(* CODESYS project Elevator.project

Project tree, tasks and I/O mapping:
  Device : Elmo Platinum Maestro, Elmo Motion Control, version 1.0.0.2
    application Application
      libraries: Standard, * (System); VisuDialogs, * (System)
      task MainTask (cyclic, interval t#20ms, priority 1) calls PLC_PRG
      task VISU_TASK (cyclic, interval 100 ms, priority 31) calls VisuElems.Visu_Prg
      program PLC_PRG [ST]
      visualisation Visualization
      visualisation Elevator
      01_Enumerator/
        data type eFloor
      02_Structure/
        data type stElevator
        data type stFloor
      03_Module/
        function block FB_Elevator [ST]: M_SpecialFloorSelect, pSpecialFloor, M_DoorStatus, M_ElevatorType, M_FindFloor, M_ElevatorMove, M_ElevatorSelect, M_ElevatorButtonDisable, M_FloorMove
        function block FB_FreightElevator [ST]: pSpecialFloor
        function block FB_Floor [ST]
        function F_RandElevator [ST]
      04_Component/
      visualisation Floor
      global variables GVL_Random
    Elmo_Master_Device : Elmo Master Device, Elmo, version 1.0.0.2
  libraries: VisuSymbols, 3.5.10.0 (System)
  text list GlobalTextList
*)

// Device/Application/02_Structure/stElevator
TYPE stElevator :
STRUCT
	sElMove: STRING;
	xFloor1: BOOL;
	
	xFloor2: BOOL;
	
	xFloor3: BOOL;
	
	xFloor4: BOOL;
	
	xFloor5: BOOL;
	
	xSpecialFloor: BOOL;
	xSpecialLight: BOOL;
	sSpecialFloorText: STRING;
	xInvisibleLamp: BOOL;
	
	xOpen: BOOL;
	xClose: BOOL;
	sDoorStatus: STRING;
	//trig_Door: r_trig;
	//trig_CloseDoor: r_trig;
	sElevatorType: STRING;
	iElevatorMove: INT;
	
	sElevatorFloor: STRING;
END_STRUCT
END_TYPE

// Device/Application/02_Structure/stFloor
TYPE stFloor :
STRUCT
	sFloor: STRING;
	iPeople: INT;
	iPeopleCurrent: INT;
	xCall: BOOL;
END_STRUCT
END_TYPE

// Device/Application/01_Enumerator/eFloor
{attribute 'qualified_only'}
{attribute 'strict'}
TYPE eFloor :
(
	F1 := 0,
	F2 := -475,
	F3 := -935,
	F4 := -1375,
	F5 := -1800
);
END_TYPE

// Device/Application/GVL_Random
{attribute 'qualified_only'}
VAR_GLOBAL
	g_seed : INT := 107;
END_VAR

// Device/Application/PLC_PRG
PROGRAM PLC_PRG
VAR
	stFloorData: ARRAY[1..uiFloors] OF stFloor;
	fbFloor: ARRAY[1..uiFloors] OF FB_Floor;
	iFloor: INT;
	stFreightFloor: stFloor;
	iRandFloor: int;
	
	stElevatorData: ARRAY[1..uiElevators] OF stElevator;
	fbElevator: ARRAY[1..uiElevators] OF FB_Elevator;
	iElevator: INT;
	stFreightElevator: stElevator;
	fbFreightElevator: FB_FreightElevator;
	
	xRandElevator: BOOL;
END_VAR

VAR CONSTANT
	uiFloors: UINT:= 5;
	uiElevators: UINT:= 3;
END_VAR

FOR iFloor:=1 TO uiFloors BY 1 DO
	stFloorData[iFloor].sFloor := concat(str1:='F',str2:=INT_TO_STRING(iFloor));
	stFloorData[iFloor].iPeopleCurrent := stFloorData[iFloor].iPeople;
	
	//IF stFloorData[iFloor].xCall = TRUE THEN
		//iRandFloor := F_RandElevator();
		//stElevatorData[iRandFloor]
		//IF NOT xRandElevator THEN
			//iRandFloor := F_RandElevator();
			//xRandElevator := TRUE;
		//END_IF
		iRandFloor := fbElevator[iFloor].M_ElevatorSelect(is_Floor := stFloorData[iFloor].sFloor,ist_Elevator:=stElevatorData);
		//stElevatorData[iRandFloor].sElMove := fbElevator[iRandFloor].os_ElMove;
		fbElevator[iRandFloor].M_ElevatorMove(is_Floor := stFloorData[iFloor].sFloor,iElMove := stElevatorData[iRandFloor].iElevatorMove,xElevatorMove := stFloorData[iFloor].xCall);
		//stFloorData[iFloor].xCall := FALSE;
	//END_IF
END_FOR

stFreightFloor.sFloor := 'B1';
stFreightFloor.iPeopleCurrent := stFreightFloor.iPeople;
//iRandFloor := F_RandElevator();


FOR iElevator:= 1 TO uiElevators BY 1 DO
	
    stElevatorData[iElevator].sElMove := fbElevator[iElevator].os_ElMove;
	stElevatorData[iElevator].sSpecialFloorText := fbElevator[iElevator].pSpecialFloor;
	fbElevator[iElevator].ix_FloorButton := stElevatorData[iElevator].xSpecialFloor;
	stElevatorData[iElevator].xSpecialLight := fbElevator[iElevator].M_SpecialFloorSelect();
	
	fbElevator[iElevator].M_DoorStatus(ix_Open:=stElevatorData[iElevator].xOpen,ix_Close:= stElevatorData[iElevator].xClose);
	stElevatorData[iElevator].sDoorStatus := fbElevator[iElevator].os_DoorStatus;
	stElevatorData[iElevator].xOpen := fbElevator[iElevator].ox_Door;
	stElevatorData[iElevator].xClose := NOT fbElevator[iElevator].ox_Door;
	fbElevator[iElevator].M_ElevatorType(is_SpecialFloorText:= stElevatorData[iElevator].sSpecialFloorText);
	stElevatorData[iElevator].sElevatorType := fbElevator[iElevator].os_ElevatorType;
	//IF(stElevatorData[iElevator].iElevatorMove <> -1800) THEN
	  //stElevatorData[iElevator].iElevatorMove := stElevatorData[iElevator].iElevatorMove-1;
    //END_IF
	//IF(stElevatorData[iElevator].xFloor1 = TRUE) THEN
		//IF stElevatorData[iElevator].iElevatorMove < -475 THEN
	      //stElevatorData[iElevator].iElevatorMove := stElevatorData[iElevator].iElevatorMove+1;
        //END_IF

        //IF stElevatorData[iElevator].iElevatorMove > -475 THEN
	      //stElevatorData[iElevator].iElevatorMove := stElevatorData[iElevator].iElevatorMove-1;
        //END_IF
	//END_IF
	fbElevator[iElevator].M_ElevatorButtonDisable(xF1:= stElevatorData[iElevator].xFloor1, xF2:= stElevatorData[iElevator].xFloor2, xF3:= stElevatorData[iElevator].xFloor3, xF4:= stElevatorData[iElevator].xFloor4, xF5:= stElevatorData[iElevator].xFloor5);
	fbElevator[iElevator].M_FloorMove(xFloorButton := stElevatorData[iElevator].xFloor1,is_Floor:= 'F1',iElMove := stElevatorData[iElevator].iElevatorMove);
	fbElevator[iElevator].M_FloorMove(xFloorButton := stElevatorData[iElevator].xFloor2,is_Floor:= 'F2',iElMove := stElevatorData[iElevator].iElevatorMove);
	fbElevator[iElevator].M_FloorMove(xFloorButton := stElevatorData[iElevator].xFloor3,is_Floor:= 'F3',iElMove := stElevatorData[iElevator].iElevatorMove);
	fbElevator[iElevator].M_FloorMove(xFloorButton := stElevatorData[iElevator].xFloor4,is_Floor:= 'F4',iElMove := stElevatorData[iElevator].iElevatorMove);
	fbElevator[iElevator].M_FloorMove(xFloorButton := stElevatorData[iElevator].xFloor5,is_Floor:= 'F5',iElMove := stElevatorData[iElevator].iElevatorMove);
	stElevatorData[iElevator].sElevatorFloor := fbElevator[iElevator].M_FindFloor(iElMove:= stElevatorData[iElevator].iElevatorMove);
	
END_FOR

stFreightElevator.sSpecialFloorText := fbFreightElevator.pSpecialFloor;
stFreightElevator.xInvisibleLamp := TRUE;
fbFreightElevator.M_DoorStatus(ix_Open:=stFreightElevator.xOpen,ix_Close:= stFreightElevator.xClose);
stFreightElevator.sDoorStatus := fbFreightElevator.os_DoorStatus;
stFreightElevator.xOpen := fbFreightElevator.ox_Door;
stFreightElevator.xClose := NOT fbFreightElevator.ox_Door;
fbFreightElevator.M_ElevatorType(is_SpecialFloorText:= stFreightElevator.sSpecialFloorText);
stFreightElevator.sElevatorType := fbFreightElevator.os_ElevatorType;
//IF(stFreightElevator.iElevatorMove <> -1400) THEN
	//stFreightElevator.iElevatorMove := stFreightElevator.iElevatorMove-1;
//END_IF

END_PROGRAM

// Device/Application/03_Module/F_RandElevator
FUNCTION F_RandElevator : INT
VAR_INPUT
END_VAR
VAR
END_VAR

GVL_Random.g_seed := GVL_Random.g_seed * 41 + 17;

IF GVL_Random.g_seed < 0 THEN
    GVL_Random.g_seed := -GVL_Random.g_seed;
END_IF;

F_RandElevator := (GVL_Random.g_seed MOD 3) + 1;

END_FUNCTION

// Device/Application/03_Module/FB_Floor
FUNCTION_BLOCK FB_Floor
VAR_INPUT
END_VAR
VAR_OUTPUT
END_VAR
VAR
END_VAR

END_FUNCTION_BLOCK

// Device/Application/03_Module/FB_Elevator
FUNCTION_BLOCK FB_Elevator
VAR_INPUT
	ix_FloorButton: BOOL;
	ix_Open: BOOL;
	ix_Close: BOOL;
	is_SpecialFloorText: STRING;
	iElMove: INT;
	is_Floor: STRING;
END_VAR
VAR_OUTPUT
	ox_FloorLight: BOOL;
	ox_Door: BOOL;
	os_DoorStatus: STRING;
	os_ElevatorType: STRING;
	os_ElMove: STRING;
END_VAR
VAR
	sSpecialFloorText: STRING;
	trig_Door: r_trig;
	trig_CloseDoor: r_trig;
	iChangeString: INT;
	iFloorValue: eFloor;
	xElevatorMove: BOOL;
	a:INT;
	b:INT;
	c:INT;
	
	d1:INT;
	d2:INT;
	d3:INT;
	mindiff: INT;
	req: INT;
	xFloorButton: BOOL;
	xF1: BOOL;
	xF2: BOOL;
	xF3: BOOL;
	xF4: BOOL;
	xF5: BOOL;
END_VAR

METHOD M_SpecialFloorSelect : BOOL
VAR_INPUT
END_VAR
IF ix_FloorButton=TRUE THEN
	M_SpecialFloorSelect := TRUE;
ELSE
	M_SpecialFloorSelect := FALSE;
END_IF
END_METHOD

PROPERTY pSpecialFloor : STRING
GET
pSpecialFloor := 'EMG';
END_GET
END_PROPERTY

METHOD M_DoorStatus : BOOL
VAR_INPUT
	ix_Open: BOOL;
	ix_Close: BOOL;
END_VAR
trig_Door(clk:=ix_Open);
trig_CloseDoor(clk:=ix_Close);

IF trig_CloseDoor.Q THEN
	ox_Door := FALSE;
ELSIF trig_Door.Q THEN
	ox_Door:= TRUE;
END_IF

IF ox_Door THEN
	os_DoorStatus := 'OPEN';
ELSE
	os_DoorStatus := 'CLOSED';
END_IF
END_METHOD

METHOD M_ElevatorType : STRING
VAR_INPUT
	is_SpecialFloorText: STRING;
END_VAR
IF is_SpecialFloorText = 'EMG' THEN
	os_ElevatorType := 'Max 3 People';
ELSIF is_SpecialFloorText = 'B1' THEN
	os_ElevatorType := 'Max 5 People';
END_IF
END_METHOD

METHOD M_FindFloor : STRING
VAR_INPUT
	iElMove: INT;
END_VAR
IF iElMove <= 0 AND iElMove >= -150 THEN
	M_FindFloor := 'F1';

ELSIF iElMove <= -475 AND iElMove >= -650 THEN
	M_FindFloor := 'F2';

ELSIF iElMove <= -935 AND iElMove >= -1150 THEN
	M_FindFloor := 'F3';

ELSIF iElMove <= -1375 AND iElMove >= -1550 THEN
	M_FindFloor := 'F4';

ELSIF iElMove >= -1800  AND iElMove <= -1650 THEN
	M_FindFloor := 'F5';
	
ELSE
	M_FindFloor := 'Moving';
END_IF
END_METHOD

METHOD M_ElevatorMove : STRING
VAR_INPUT
	is_Floor: STRING;
END_VAR
VAR_IN_OUT
    iElMove  : INT;   // now the value can change outside
	xElevatorMove : BOOL;
END_VAR
IF is_Floor = 'F1' THEN
    iFloorValue := eFloor.F1;
ELSIF is_Floor = 'F2' THEN
    iFloorValue := eFloor.F2;
ELSIF is_Floor = 'F3' THEN
    iFloorValue := eFloor.F3;
ELSIF is_Floor = 'F4' THEN
    iFloorValue := eFloor.F4;
ELSIF is_Floor = 'F5' THEN
    iFloorValue := eFloor.F5;
END_IF

IF xElevatorMove = TRUE THEN
	IF iElMove < iFloorValue THEN
	  iElMove := iElMove + 1;
	  os_ElMove := 'DOWN';
    END_IF

    IF iElMove > iFloorValue THEN
	   iElMove := iElMove - 1;
	   os_ElMove := 'UP';
    END_IF
	
	IF iElMove = iFloorValue THEN
	   //iElMove := iElMove - 1;
	   xElevatorMove := FALSE;
	   os_ElMove := 'UP/DOWN';
    END_IF
END_IF


//IF iElMove = iFloorValue THEN
	//xElevatorMove := FALSE;
//END_IF
END_METHOD

METHOD M_ElevatorSelect : INT
VAR_INPUT
	is_Floor: STRING;
	ist_Elevator: ARRAY[1..3] OF stElevator;
END_VAR
IF is_Floor = 'F1' THEN
    iFloorValue := eFloor.F1;
ELSIF is_Floor = 'F2' THEN
    iFloorValue := eFloor.F2;
ELSIF is_Floor = 'F3' THEN
    iFloorValue := eFloor.F3;
ELSIF is_Floor = 'F4' THEN
    iFloorValue := eFloor.F4;
ELSIF is_Floor = 'F5' THEN
    iFloorValue := eFloor.F5;
END_IF;

a := ist_Elevator[1].iElevatorMove;
b := ist_Elevator[2].iElevatorMove;
c := ist_Elevator[3].iElevatorMove;

req:=iFloorValue;
d1 := ABS(a - req);
d2 := ABS(b - req);
d3 := ABS(c - req);


minDiff := MIN(d1, MIN(d2, d3));

IF minDiff = d1 THEN
	M_ElevatorSelect := 1;
ELSIF mindiff = d2 THEN
	M_ElevatorSelect := 2;
ELSE
	M_ElevatorSelect := 3;
END_IF
END_METHOD

METHOD M_ElevatorButtonDisable
VAR_INPUT
END_VAR
VAR_IN_OUT
	xF1: BOOL;
	xF2: BOOL;
	xF3: BOOL;
	xF4: BOOL;
	xF5: BOOL;
END_VAR
IF (xF1 = TRUE) OR NOT (xF1 OR xF2 OR xF3 OR xF4 OR xF5) THEN
	xF1 := TRUE;
	xF2 := FALSE;
	xF3 := FALSE;
	xF4 := FALSE;
	XF5 := FALSE;
END_IF

IF (xF2 = TRUE) OR NOT (xF1 OR xF2 OR xF3 OR xF4 OR xF5) THEN
	xF2 := TRUE;
	xF1 := FALSE;
	xF3 := FALSE;
	xF4 := FALSE;
	XF5 := FALSE;
END_IF

IF (xF3 = TRUE) OR NOT (xF1 OR xF2 OR xF3 OR xF4 OR xF5) THEN
	xF3 := TRUE;
	xF1 := FALSE;
	xF2 := FALSE;
	xF4 := FALSE;
	XF5 := FALSE;
END_IF

IF (xF4 = TRUE) OR NOT (xF1 OR xF2 OR xF3 OR xF4 OR xF5) THEN
	xF4 := TRUE;
	xF1 := FALSE;
	xF2 := FALSE;
	xF3 := FALSE;
	XF5 := FALSE;
END_IF

IF (xF5 = TRUE) OR NOT (xF1 OR xF2 OR xF3 OR xF4 OR xF5) THEN
	xF5 := TRUE;
	xF1 := FALSE;
	xF2 := FALSE;
	xF3 := FALSE;
	XF4 := FALSE;
END_IF
END_METHOD

METHOD M_FloorMove
VAR_INPUT
	is_Floor: STRING;
END_VAR
VAR_IN_OUT
    iElMove  : INT;   // now the value can change outside
	//xElevatorMove : BOOL;
	xFloorButton: BOOL;
END_VAR
IF is_Floor = 'F1' THEN
    iFloorValue := eFloor.F1;
ELSIF is_Floor = 'F2' THEN
    iFloorValue := eFloor.F2;
ELSIF is_Floor = 'F3' THEN
    iFloorValue := eFloor.F3;
ELSIF is_Floor = 'F4' THEN
    iFloorValue := eFloor.F4;
ELSIF is_Floor = 'F5' THEN
    iFloorValue := eFloor.F5;
END_IF;


IF(xFloorButton = TRUE) THEN
	IF iElMove < iFloorValue THEN
	  iElMove := iElMove + 1;
	  os_ElMove := 'DOWN';
    END_IF

    IF iElMove > iFloorValue THEN
	   iElMove := iElMove - 1;
	   os_ElMove := 'UP';
    END_IF
	
	IF iElMove = iFloorValue THEN
	   xFloorButton := FALSE;
	   os_ElMove := 'UP/DOWN';
    END_IF
END_IF
END_METHOD

END_FUNCTION_BLOCK

// Device/Application/03_Module/FB_FreightElevator
FUNCTION_BLOCK FB_FreightElevator EXTENDS FB_Elevator
VAR_INPUT
END_VAR
VAR_OUTPUT
END_VAR
VAR
END_VAR

SUPER^();

PROPERTY pSpecialFloor : STRING
GET
pSpecialFloor := 'B1';
END_GET
END_PROPERTY

END_FUNCTION_BLOCK

// Device/Application/Visualization
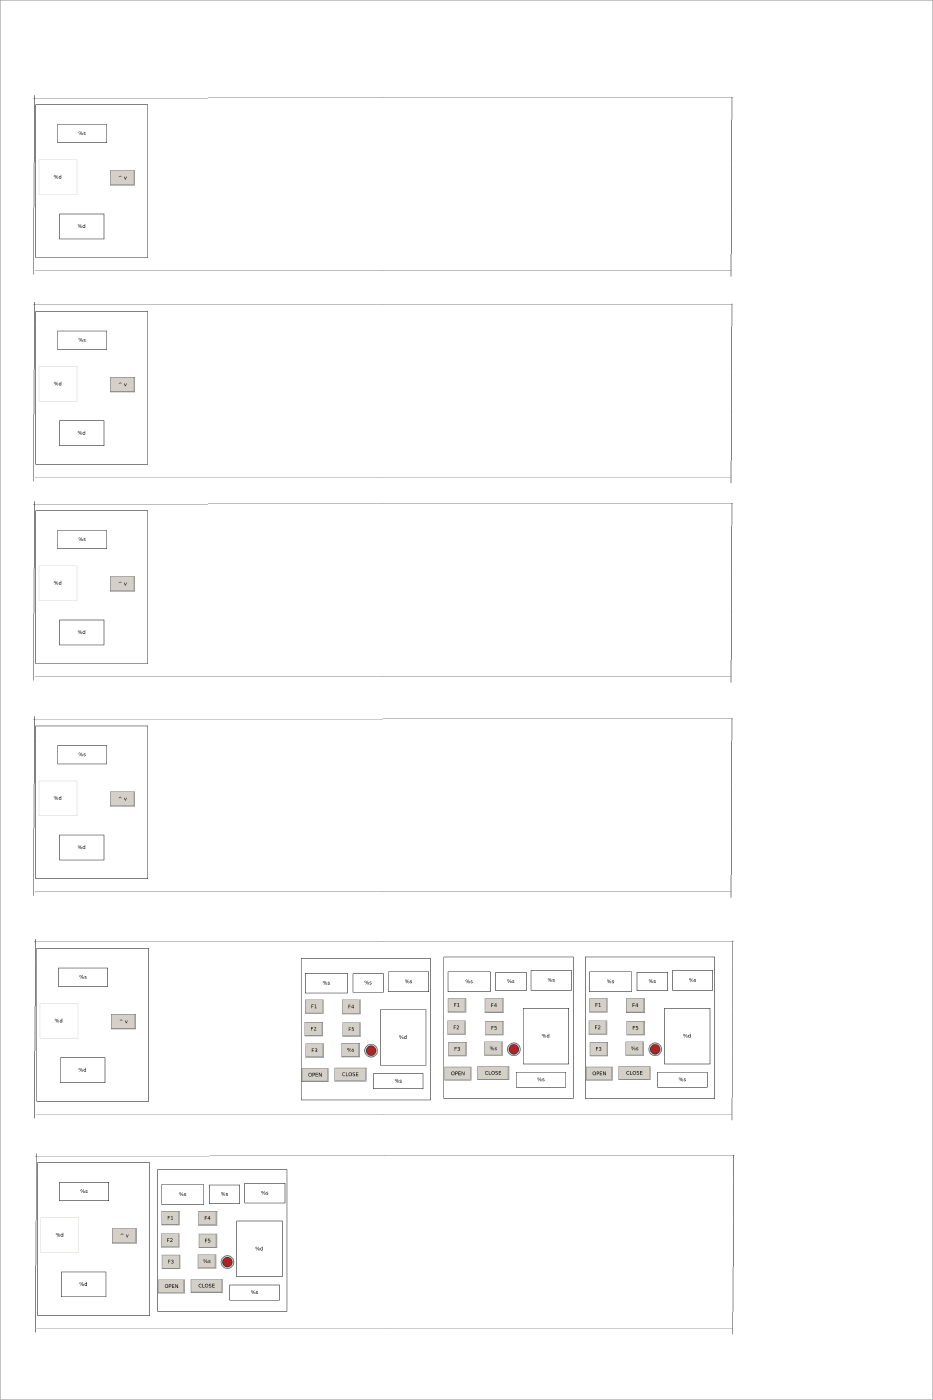
VISUALIZATION Visualization  // 2000x3000
    Frame (75,2464 1501x400)
        shows Floor(stFloorVisu := PLC_PRG.stFreightFloor)
    Frame (337,2505 278x304)
        shows Elevator(stElevatorVisu := PLC_PRG.stFreightElevator)
    Frame (71,1067 1501x400)
        shows Floor(stFloorVisu := PLC_PRG.stFloorData[3])
    Frame (71,640 1501x400)
        shows Floor(stFloorVisu := PLC_PRG.stFloorData[4])
    Frame (71,197 1501x400)
        shows Floor(stFloorVisu := PLC_PRG.stFloorData[5])
    Frame (73,2005 1501x400)
        shows Floor(stFloorVisu := PLC_PRG.stFloorData[1])
    Frame (71,1528 1501x400)
        shows Floor(stFloorVisu := PLC_PRG.stFloorData[2])
    Frame (645,2052 278x304)
        shows Elevator(stElevatorVisu := PLC_PRG.stElevatorData[1])
    Frame (951,2049 278x304)
        shows Elevator(stElevatorVisu := PLC_PRG.stElevatorData[2])
    Frame (1254,2049 278x304)
        shows Elevator(stElevatorVisu := PLC_PRG.stElevatorData[3])
END_VISUALIZATION

// Device/Application/Elevator
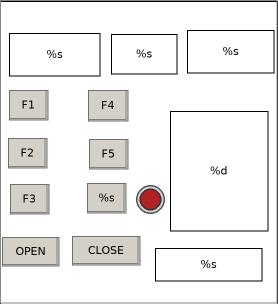
VISUALIZATION Elevator  // 278x304
VAR_IN_OUT
	stElevatorVisu : stElevator;
END_VAR
    Group (0,1 278x304)
        p2738717112: stElevatorVisu.iElevatorMove
        Rectangle (0,0 278x304)
        Rectangle (155,247 107x33), "%s", text variable: stElevatorVisu.sDoorStatus
        Button (72,235 68x29), "CLOSE"
            toggle stElevatorVisu.xClose
        Button (2,236 57x29), "OPEN"
            toggle stElevatorVisu.xOpen
        Button (10,183 39x30), "F3"
            toggle stElevatorVisu.xFloor3
        Button (87,182 39x30), "%s", text variable: stElevatorVisu.sSpecialFloorText
            toggle stElevatorVisu.xSpecialFloor
        Lamp1 (134,181 33x35), variable: stElevatorVisu.xSpecialLight, invisible if: stElevatorVisu.xInvisibleLamp, style: Lamp-Lamp1-Red
        RoundedRectangle (170,110 98x120), "%d"
        Button (89,138 39x30), "F5"
            toggle stElevatorVisu.xFloor5
        Button (8,137 39x30), "F2"
            toggle stElevatorVisu.xFloor2
        Button (9,89 39x30), "F1"
            toggle stElevatorVisu.xFloor1
        Button (88,89 40x31), "F4"
            toggle stElevatorVisu.xFloor4
        Rectangle (9,32 91x43), "%s", text variable: stElevatorVisu.sElMove
        Rectangle (111,33 66x40), "%s", text variable: stElevatorVisu.sElevatorFloor
        Rectangle (187,29 87x43), "%s", text variable: stElevatorVisu.sElevatorType
END_VISUALIZATION

// Device/Application/Floor
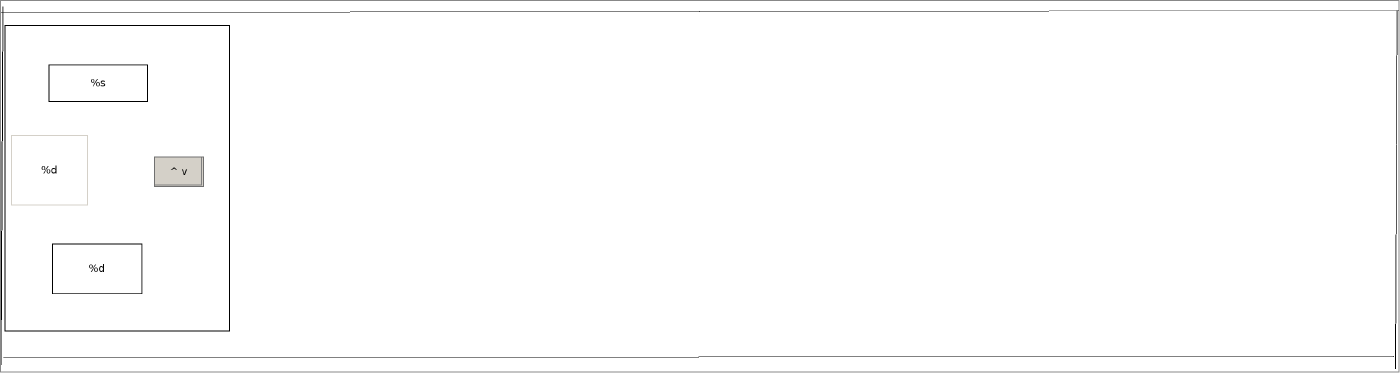
VISUALIZATION Floor  // 1501x400
VAR_IN_OUT
	stFloorVisu : stFloor;
END_VAR
    Line (1,391) (3,7)
    Line (0,13) (1499,11)
    Rectangle (5,27 241x328)
    Textfield (12,145 82x75), "%d", text variable: stFloorVisu.iPeople
        OnMouseClick: write the text variable via VisuDialogs.Numpad
    RoundedRectangle (52,69 106x40), "%s", text variable: stFloorVisu.sFloor
    RoundedRectangle (56,261 96x54), "%d", text variable: stFloorVisu.iPeopleCurrent
    Line (4,383) (1494,382)
    Line (1496,395) (1498,11)
    Button (165,168 53x32), "^ v"
        toggle stFloorVisu.xCall
END_VISUALIZATION
